Universal Robots PolyScope program: hmi_chart_monitoring.urp

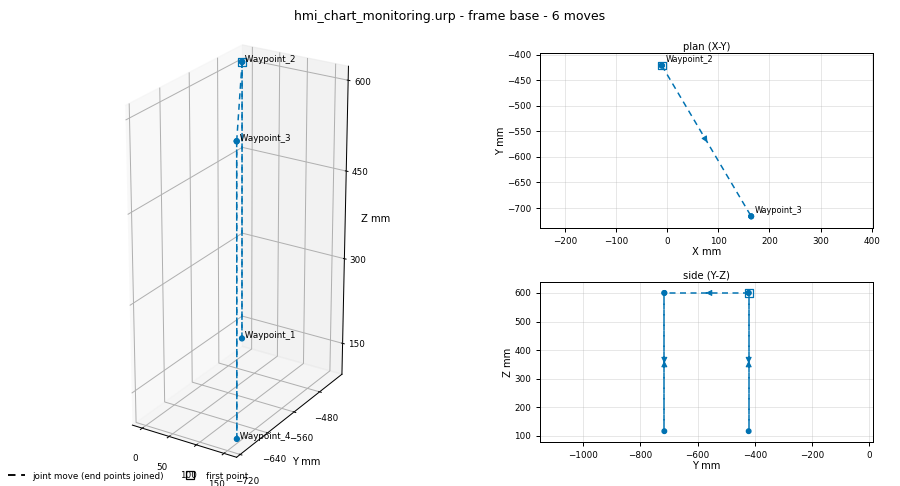
[picture p0: tool path of hmi_chart_monitoring.urp in frame base, 6 of 6 moves have a stored position in this frame; points joined in program order, loops and branches not executed]
Program chart (installation=default directory=/home/ur/ursim-current/programs createdIn=5.14.0 lastSavedIn=5.14.0 robotSerialNumber=20195299999)
Calibrated DH parameters: a=[0, -0.6127, -0.57155, 0, 0, 0]; d=[0.1807, 0, 0, 0.17415, 0.11985, 0.11655]; alpha=[1.570796, 0, 0, 1.570796, -1.570796, 0]; deltaTheta=[0, 0, 0, 0, 0, 0]
InitVariablesNode
BeforeStart
  a := 1.0
  b := 2.0
  c := 3.0
Robot Program (runOnlyOnce=false)
  Script file /home/ur/ursim-current/programs/update_data.script
    | j1 = 0
    | j2 = 0
    | j3 = 0
    | j4 = 0
    | j5 = 0
    | j6 = 0
    | 
    | x = 0
    | y = 0
    | z = 0
    | 
    | t1 = 0
    | t2 = 0
    | t3 = 0
    | t4 = 0
    | t5 = 0
    | t6 = 0
    | 
    | temp1 = 0.0
    | temp2 = 0.0
    | temp3 = 0.0
    | temp4 = 0.0
    | temp5 = 0.0
    | temp6 = 0.0
    | 
    | s1 = 0
    | s2 = 0
    | s3 = 0
    | s4 = 0
    | s5 = 0
    | s6 = 0
    | 
    | t = 0
    | 
    | distance = 1
    | max_distance = 0
    | 
    | thread update():
    |     while True:
    |         joints = get_actual_joint_positions()
    |         j1 = joints[0]
    |         j2 = joints[1]
    |         j3 = joints[2]
    |         j4 = joints[3]
    |         j5 = joints[4]
    |         j6 = joints[5]
    | 
    |     	tcp = get_actual_tcp_pose()
    |     	x = tcp[0]
    |     	y = tcp[1]+1
    |     	z = tcp[2]
    |     	sync()
    | 
    |     	torques = get_joint_torques()
    |     	#t1 = norm(torques[0])
    |         #t2 = norm(torques[1])
    |         #t3 = norm(torques[2])
    |         #t4 = norm(torques[3])
    |         #t5 = norm(torques[4])
    |         #t6 = norm(torques[5])
    | 
    |         t1 = norm(joints[0])*2 + random()
    |         t2 = norm(joints[1])*2 + random()
    |         t3 = norm(joints[2])*2 + random()
    |         t4 = norm(joints[3])*2 + random()
    |         t5 = norm(joints[4])*2 + random()
    |         t6 = norm(joints[5])*2 + random()
    |         sync()
    | 
    |         #temp1 = get_joint_temp(0)
    |         #temp2 = get_joint_temp(1)
    |         #temp3 = get_joint_temp(2)
    |         #temp4 = get_joint_temp(3)
    |         #temp5 = get_joint_temp(4)
    |         #temp6 = get_joint_temp(5)
    | 
    |         temp1 = 60 + sin(t*2)*5*random()
    |         temp2 = 75 + sin(t*3)*5*random()
    |         temp3 = 55 + sin(t*4)*5*random()
    |         temp4 = 50 + sin(t*4)*3*random()
    |         temp5 = 60 + sin(t*4)*3*random()
    |         temp6 = 55 + sin(t*4)*3*random()
    |         t = t + 0.01
    |         sync()
    | 
    |         speed = get_actual_joint_speeds()
    |         s1 = norm(speed[0])
    |         s2 = norm(speed[1])
    |         s3 = norm(speed[2])
    |         s4 = norm(speed[3])
    |         s5 = norm(speed[4])
    |         s6 = norm(speed[5])
    | 
    | 
    |     end
    | end
    | 
    | run update()
  URCap HMI (Robpod HMI URcap, Robpod Cloud) dataModel(robpod.hmi.selected=/home/ur/ursim-current/programs/monitor_hmi.hmi)
  Loop Forever
    MoveJ speed 60 deg/s, acceleration 80 deg/s^2 (useActiveTCP=true) feature=Base
      Set DigitalOutput pin=digital_out[1]; digitalValue=1
      Waypoint Waypoint_2: motionParameters(jointSpeed=1.745329 jointAcceleration=1.396263 cartesianSpeed=0.25 cartesianAcceleration=1.2); TCP in base x=-10.381 y=-421.477 z=600 mm, rx=0.6883 ry=-2.9936 rz=0.0781 rad; joints [-65.659, -58.977, -120.42, -88.522, 85.558, -1.638] deg; TCP offset x=0 y=0 z=0 mm, rx=0 ry=0 rz=0 rad
      Set DigitalOutput pin=digital_out[1]; digitalValue=0
      Waypoint Waypoint_1: motionParameters(jointSpeed=1.745329 jointAcceleration=1.396263 cartesianSpeed=0.25 cartesianAcceleration=1.2); TCP in base x=-10.381 y=-421.477 z=116.645 mm, rx=3.019 ry=0.6489 rz=-0.1053 rad; joints [-65.659, -100.849, -154.929, -12.141, 85.558, 180] deg; TCP offset x=0 y=0 z=0 mm, rx=0 ry=0 rz=0 rad
      Set DigitalOutput pin=digital_out[2]; digitalValue=0
      Set DigitalOutput pin=digital_out[0]; digitalValue=1
      Waypoint Waypoint_2: motionParameters(jointSpeed=1.745329 jointAcceleration=1.396263 cartesianSpeed=0.25 cartesianAcceleration=1.2); TCP in base x=-10.381 y=-421.477 z=600 mm, rx=0.6883 ry=-2.9936 rz=0.0781 rad; joints [-65.659, -58.977, -120.42, -88.522, 85.558, -1.638] deg; TCP offset x=0 y=0 z=0 mm, rx=0 ry=0 rz=0 rad
      Set DigitalOutput pin=digital_out[3]; digitalValue=1
      Waypoint Waypoint_3: TCP in base x=164.342 y=-716.299 z=600 mm, rx=3.0025 ry=0.7291 rz=-0.1074 rad; joints [-62.628, -92.087, -96.032, -80.038, 85.454, -180] deg; TCP offset x=0 y=0 z=0 mm, rx=0 ry=0 rz=0 rad
      Set DigitalOutput pin=digital_out[3]; digitalValue=0
      Waypoint Waypoint_4: motionParameters(jointSpeed=1.745329 jointAcceleration=1.396263 cartesianSpeed=0.25 cartesianAcceleration=1.2); TCP in base x=164.342 y=-716.299 z=116.645 mm, rx=0.6883 ry=-2.9936 rz=0.0781 rad; joints [-62.628, -118.609, -120.346, -29.203, 85.454, 1.4] deg; TCP offset x=0 y=0 z=0 mm, rx=0 ry=0 rz=0 rad
      Set DigitalOutput pin=digital_out[0]; digitalValue=0
      Waypoint Waypoint_3: motionParameters(jointSpeed=1.745329 jointAcceleration=1.396263 cartesianSpeed=0.25 cartesianAcceleration=1.2); TCP in base x=164.342 y=-716.299 z=600 mm, rx=3.0025 ry=0.7291 rz=-0.1074 rad; joints [-62.628, -92.087, -96.032, -80.038, 85.454, -180] deg; TCP offset x=0 y=0 z=0 mm, rx=0 ry=0 rz=0 rad
      Set DigitalOutput pin=digital_out[2]; digitalValue=1
